TYPE Pers_data :
STRUCT
    Name : STRING[25];
    Firstname : STRING[25];
    Gender : STRING[10]; // 'Male' of 'Female'
    Age : INT;
    Address : STRING[55];
END_STRUCT
END_TYPE

(* stored: Version 1.1.0.1, ProductVersion 3.1.4024.12
   DUT Pers_data: Id {c8acbf6d-bb0b-406a-a6e9-41d970864180} *)
